// TIA Portal project "Project_WinCCRT" (V17)

(* hardware
DEVICE "S7-1500/ET200MP station_1"  S7-1500 station
   slot 0: "Rail_0"  Rack  6ES7 590-1***0-0AA0
   slot 1: "PLC_PROCESS_LINE"  CPU 1511-1 PN  6ES7 511-1AK02-0AB0  V2.9
      slot 3: "CPU display_1"  6ES7591-1AA00-0AA0
      slot 32768: "PROFINET interface_1"  X1
         slot 32769: "Port_1"  X1 P1
         slot 32770: "Port_2"  X1 P2
      slot 34817: "Virtual CP interface port_1"  Virtual CP interface port  Virtual CP interface port
DEVICE "PC_STATION"  SIMATIC PC station
   slot 0: "PC station"  Rail  SIMATIC PC-Station  V1.0
      slot 125: "Stationmanager"  Station_Manager  V6.0.4
   slot 1: "IE general_1"  IE General  IE_CP  V8.2.0
      slot 1: "PROFINET interface"  IEGeneral.Interface.8.2.0
   slot 2: "HMI_RT_1"  WinCC RT Professional  6AV2 105-0xxxx-xxxx  17.0.0.0
*)

// ===== PLC "PLC_PROCESS_LINE"  CPU 1511-1 PN =====

VAR_GLOBAL   // PLC tag table "Motor_P101"
   "P101_START_PB" AT %I0.0 : Bool;   // HMI start command
   "P101_STOP_PB" AT %I0.1 : Bool;   // HMI stop command
   "P101_RUN_CMD" AT %Q0.2 : Bool;   // Motor running memory
   "P101_PERMISSIVE_OK" AT %I0.3 : Bool;   // All interlocks healthy
   "P101_TRIP_ACTIVE" AT %I0.4 : Bool;   // Motor/VFD Trip
   "P101_RUNNING" AT %Q0.6 : Bool;
   "P101_FAULT" AT %Q0.7 : Bool;
   "CMD_P101_Start" AT %M1.0 : Bool;
   "CMD_P101_Stop" AT %M1.1 : Bool;
   "CMD_P101_Auto" AT %M1.2 : Bool;
   "CMD_P101_Reset" AT %M1.3 : Bool;
   "P101_RESET_FAULT" AT %I1.0 : Bool;
   "P101_AUTO_MODE" AT %I1.1 : Bool;
END_VAR

DATA_BLOCK "DB_Motor_P101"   // DB1
{ S7_Optimized_Access := 'TRUE' }
VERSION : 0.1
// stored: InstanceOfName FB_motor
"FB_motor"
BEGIN
END_DATA_BLOCK

FUNCTION_BLOCK "FB_motor"   // FB1, LAD
{ S7_Optimized_Access := 'TRUE' }
VERSION : 0.1
   VAR_INPUT
      start_cmd : Bool;   // start request (HMI/Auto logic)
      stop_cmd : Bool;   // stop request
      permissive_ok : Bool;   // all interlocks - healthy
      reset_fault : Bool;   // reset fault input
      trip_input : Bool;   // tripping input (VFD, Overloaf)
      auto_mode : Bool;   // automatic mode on
   END_VAR
   VAR_OUTPUT
      run_cmd : Bool;   // command to motor
      running : Bool;   // motor running status
      fault : Bool;   // latched fault
   END_VAR
   VAR_IN_OUT
      "EN_S/R_RELAY" : Bool := true;
   END_VAR
   VAR
      run_latch : Bool;
   END_VAR
BEGIN

REGION Network 1: Motor running memory
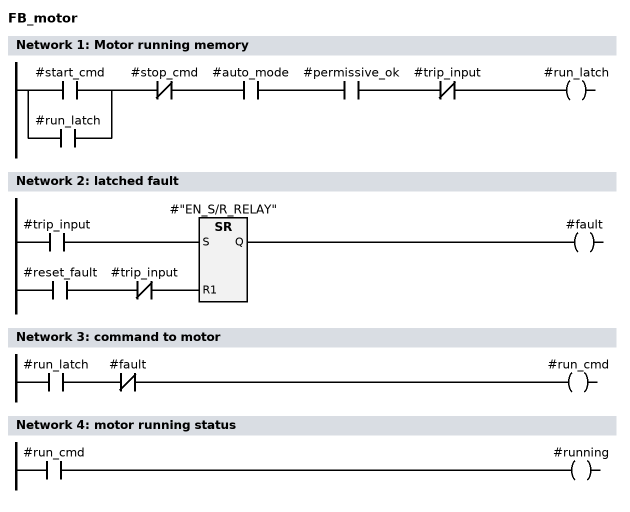
   RUNG wire#powerrail
      Contact( #start_cmd )
      wire#w1
      I_Contact( #stop_cmd )
      Contact( #auto_mode )
      Contact( #permissive_ok )
      I_Contact( #trip_input )
      Coil( #run_latch )
   END_RUNG
   RUNG wire#powerrail
      Contact( #run_latch )
   END_RUNG wire#w1
   // the same network as SCL:
   #run_latch := (#start_cmd OR #run_latch) AND NOT #stop_cmd AND #auto_mode AND #permissive_ok AND NOT #trip_input;
END_REGION

REGION Network 2: latched fault
   RUNG wire#powerrail
      Contact( #trip_input )
      S_SR(operand := #"EN_S/R_RELAY", r1 := wire#w1)
      Coil( #fault )
   END_RUNG
   RUNG wire#powerrail
      Contact( #reset_fault )
      I_Contact( #trip_input )
   END_RUNG wire#w1
   // the same network as SCL:
   IF #trip_input THEN
       #"EN_S/R_RELAY" := TRUE;   // SR flip-flop
   END_IF;
   IF #reset_fault AND NOT #trip_input THEN #"EN_S/R_RELAY" := FALSE; END_IF;
   #fault := #"EN_S/R_RELAY";
END_REGION

REGION Network 3: command to motor
   RUNG wire#powerrail
      Contact( #run_latch )
      I_Contact( #fault )
      Coil( #run_cmd )
   END_RUNG
   // the same network as SCL:
   #run_cmd := #run_latch AND NOT #fault;
END_REGION

REGION Network 4: motor running status
   RUNG wire#powerrail
      Contact( #run_cmd )
      Coil( #running )
   END_RUNG
   // the same network as SCL:
   #running := #run_cmd;
END_REGION
END_FUNCTION_BLOCK

ORGANIZATION_BLOCK "Main"   // OB1, LAD, ProgramCycle
TITLE = "Main Program Sweep (Cycle)"
{ S7_Optimized_Access := 'TRUE' }
VERSION : 0.1
   VAR_INPUT
      Initial_Call : Bool;   // Initial call of this OB
      Remanence : Bool;   // =True, if remanent data are available
   END_VAR
BEGIN

REGION Network 1
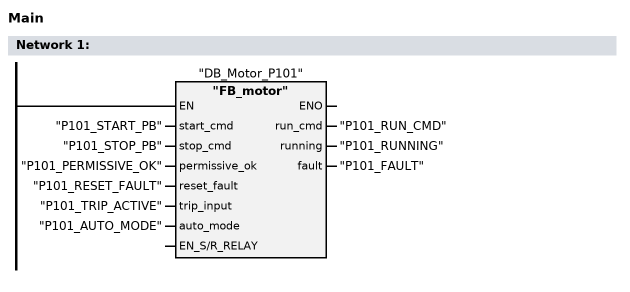
   RUNG wire#powerrail
      "DB_Motor_P101"(start_cmd := "P101_START_PB", stop_cmd := "P101_STOP_PB", permissive_ok := "P101_PERMISSIVE_OK", reset_fault := "P101_RESET_FAULT", trip_input := "P101_TRIP_ACTIVE", auto_mode := "P101_AUTO_MODE", "EN_S/R_RELAY" :=, run_cmd => "P101_RUN_CMD", running => "P101_RUNNING", fault => "P101_FAULT")
   END_RUNG
   // the same network as SCL:
   "DB_Motor_P101"(start_cmd := "P101_START_PB",   // "FB_motor"
                   stop_cmd := "P101_STOP_PB",
                   permissive_ok := "P101_PERMISSIVE_OK",
                   reset_fault := "P101_RESET_FAULT",
                   trip_input := "P101_TRIP_ACTIVE",
                   auto_mode := "P101_AUTO_MODE",
                   run_cmd => "P101_RUN_CMD",
                   running => "P101_RUNNING",
                   fault => "P101_FAULT");
END_REGION
END_ORGANIZATION_BLOCK

(* ===== HMI "HMI_RT_1" =====
system functions are stored by id; their names below are inferred from use
connection "HMI_Connection_1": S71200_TCP_IP, SCADA_S7_1500_OMS

HMI tags "Default tag table"
   "P101_START_PB" : Bool = PLC P101_START_PB AT %I0.0, 500 ms
   "P101_STOP_PB" : Bool = PLC P101_STOP_PB AT %I0.1, 500 ms
   "P101_RESET_FAULT" : Bool = PLC P101_RESET_FAULT AT %I1.0, 500 ms
   "P101_PERMISSIVE_OK" : Bool = PLC P101_PERMISSIVE_OK AT %I0.3, 500 ms
   "P101_TRIP_ACTIVE" : Bool = PLC P101_TRIP_ACTIVE AT %I0.4, 500 ms
   "P101_AUTO_MODE" : Bool = PLC P101_AUTO_MODE AT %I1.1, 500 ms
   "P101_RUNNING" : Bool = PLC P101_RUNNING AT %Q0.6, 500 ms
   "P101_RUN_CMD" : Bool = PLC P101_RUN_CMD AT %Q0.2, 500 ms
   "P101_FAULT" : Bool = PLC P101_FAULT AT %Q0.7, 500 ms

HMI tags "Tag table_1"
   "HMI_Tag_START" : Bool = PLC CMD_P101_Start AT %M1.0, 500 ms
   "HMI_Tag_STOP" : Bool = PLC CMD_P101_Stop AT %M1.1, 500 ms
   "HMI_Tag_RESET" : Bool = PLC CMD_P101_Reset AT %M1.3, 500 ms
   "HMI_Tag_PERMISSIVE" : Bool = PLC P101_PERMISSIVE_OK AT %I0.3, 500 ms
   "HMI_Tag_AUTO_MODE" : Bool = PLC CMD_P101_Auto AT %M1.2, 500 ms
   "HMI_Tag_TRIP_ACTIVE" : Bool = PLC P101_TRIP_ACTIVE AT %I0.4, 500 ms
   "HMI_Tag_RUN_CMD" : Bool = PLC P101_RUN_CMD AT %Q0.2, 500 ms
   "HMI_Tag_RUNNING" : Bool = PLC P101_RUNNING AT %Q0.6, 500 ms
   "HMI_Tag_FAULT" : Bool = PLC P101_FAULT AT %Q0.7, 500 ms

screen "Screen_1" 1024x768
   Circle "Circle_1" at 573,58 size 48x48
      BackColor <- "HMI_Tag_RUNNING"
   TextField "Text field_1" at 43,131 size 32x21; Text 'stop'
   Button "Button_2" at 149,76 size 80x30; TextOff 'Text'; PictureOff "Graphic_3"; PictureOn "Up_Arrow"
      on PressLeft: SetBit("HMI_Tag_START")
      on PressRight: ResetBit("P101_START_PB")
   TextField "Text field_2" at 43,78 size 33x21; Text 'start'
   TextField "Text field_3" at 43,191 size 36x21; Text 'reset'
   TextField "Text field_4" at 43,253 size 77x21; Text 'permissive'
   TextField "Text field_5" at 43,315 size 75x21; Text 'trip_active'
   TextField "Text field_6" at 43,377 size 82x21; Text 'auto_mode'
   TextField "Text field_7" at 449,71 size 57x21; Text 'running'
   Circle "Circle_2" at 573,143 size 48x48
      BackColor <- "HMI_Tag_RUN_CMD"
   TextField "Text field_8" at 449,156 size 61x21; Text 'run cmd'
   Circle "Circle_3" at 573,228 size 48x48
      BackColor <- "HMI_Tag_FAULT"
   TextField "Text field_9" at 449,241 size 33x21; Text 'fault'
   Button "Button_1" at 149,131 size 80x30; TextOff 'Text'; PictureOn "Up_Arrow"; PictureOff "Graphic_3"
      on PressRight: ResetBit("HMI_Tag_STOP")
      on PressLeft: SetBit("HMI_Tag_STOP")
   Button "Button_3" at 149,186 size 80x30; TextOff 'Text'; PictureOn "Up_Arrow"; PictureOff "Graphic_3"
      on PressRight: ResetBit("HMI_Tag_RESET")
      on PressLeft: SetBit("HMI_Tag_RESET")
   Button "Button_4" at 148,251 size 80x30; TextOff 'Text'; PictureOn "Up_Arrow"; PictureOff "Graphic_3"
      on PressRight: ResetBit("HMI_Tag_PERMISSIVE")
      on PressLeft: SetBit("HMI_Tag_PERMISSIVE")
   Button "Button_5" at 148,315 size 80x30; TextOff 'Text'; PictureOn "Up_Arrow"; PictureOff "Graphic_3"
      on PressRight: ResetBit("HMI_Tag_TRIP_ACTIVE")
      on PressLeft: SetBit("HMI_Tag_TRIP_ACTIVE")
   Button "Button_6" at 148,379 size 80x30; TextOff 'Text'; PictureOn "Up_Arrow"; PictureOff "Graphic_3"
      on PressRight: ResetBit("HMI_Tag_AUTO_MODE")
      on PressLeft: SetBit("HMI_Tag_AUTO_MODE")
*)